TYPE PartStatus :
STRUCT
	Status			: BOOL;
	Diameter		: LREAL;
	Rate			: LREAL;
	Torque			: LREAL;
	Operator		: STRING;
END_STRUCT
END_TYPE

(* stored: Version 1.1.0.1
   DUT PartStatus: Id {7b521bea-ede0-4568-856b-93adf4026157} *)
